// TIA Portal V17 export
// export: Created 2022-07-20T07:01:28.9858046Z, ExportSetting WithDefaults, DisplayName Totally Integrated Automation Portal, DisplayVersion V17, DisplayName TIA Portal Openness, DisplayVersion V17, DisplayName TIA Portal Version Control Interface, DisplayVersion V17, DisplayName SINAMICS Startdrive Advanced, DisplayVersion V17, DisplayName SINAMICS Startdrive G130, G150, S120, S150, SINAMICS MV, S210, DisplayVersion V17, DisplayName SINAMICS Startdrive G110M, G120, G120C, G120D, G120P, G115D, DisplayVersion V17, DisplayName STEP 7 Professional, DisplayVersion V17, DisplayName STEP 7 Safety, DisplayVersion V17, DisplayName WinCC Advanced, DisplayVersion V17
FUNCTION_BLOCK "FB10252_IfmDV2131"   // FB10252, LAD
{ S7_Optimized_Access := 'TRUE' }
VERSION : 0.1
// stored: AutoNumber false, IsIECCheckEnabled false, IsRetainMemResEnabled false, MemoryReserve 100, SetENOAutomatically false, UDAEnableTagReadback false
   VAR_INPUT
      Segment1_Color : Byte;
      Segment1_Frequency : Byte;
      BuzerActivation : Bool;
      BuzerStyle : Byte;
   END_VAR
   VAR_OUTPUT
      ButtonPressed : Bool;
      RTrigButtonPressed : Bool;
   END_VAR
   VAR_IN_OUT
      ProcessDataWordOut_0 : Word;
      ProcessDataWordIn_0 : Word;
   END_VAR
   VAR
      RTrig_ButtonPressed : R_TRIG;
      LocalSegment1_Color { S7_SetPoint := 'True'} : Byte;
   END_VAR
BEGIN

REGION Network 1 (SCL): ADAPT cOLOR CONSTANT TO THIS DV SPECIFICATION
   CASE #Segment1_Color OF
       "SEGMENT_LED_OFF": 
           #LocalSegment1_Color := 0;
       "SEGMENT_LED_BLUE" :
           #LocalSegment1_Color := 4;
       "SEGMENT_LED_GREEN" :
           #LocalSegment1_Color := 2;
       "SEGMENT_LED_TURQUOISE" :
           #LocalSegment1_Color := 6;
       "SEGMENT_LED_RED" :
           #LocalSegment1_Color := 1;
       "SEGMENT_LED_VIOLET" :
           #LocalSegment1_Color := 5;
       "SEGMENT_LED_ORANGE" :
           #LocalSegment1_Color := 3;
       "SEGMENT_LED_WHITE" :
           #LocalSegment1_Color := 7;
       "SEGMENT_LED_YELLOW" :
           #LocalSegment1_Color := 8;

       ELSE  
           #LocalSegment1_Color := 0;
   END_CASE;
END_REGION

REGION Network 2 (SCL): Segment 1
   #ProcessDataWordOut_0 := 0;
   #ProcessDataWordOut_0.%B0 := #LocalSegment1_Color OR #Segment1_Frequency;
   #ProcessDataWordOut_0.%B1 := #BuzerStyle;
   #ProcessDataWordOut_0.%X8 := #BuzerActivation;
END_REGION

REGION Network 3: Button detection
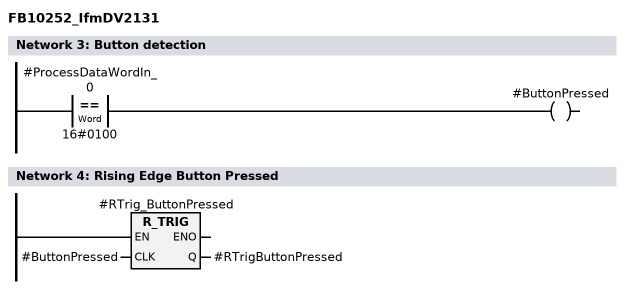
   RUNG wire#powerrail
      { S7_Templates := "SrcType := Word" } EQ_Contact(in1 := #ProcessDataWordIn_0, in2 := 16#0100)
      Coil( #ButtonPressed )
   END_RUNG
   // the same network as SCL:
   #ButtonPressed := #ProcessDataWordIn_0 = 16#0100;
END_REGION

REGION Network 4: Rising Edge Button Pressed
   RUNG wire#powerrail
      #RTrig_ButtonPressed.R_TRIG(CLK := #ButtonPressed, Q => #RTrigButtonPressed)
   END_RUNG
   // the same network as SCL:
   #RTrig_ButtonPressed(CLK := #ButtonPressed, Q => #RTrigButtonPressed);   // R_TRIG
END_REGION
END_FUNCTION_BLOCK
